FUNCTION F_RoundReal : REAL
VAR_INPUT
  rInput : REAL;
  iDecimalPlaces : INT;
END_VAR
VAR
  rOutput : REAL;
  r_Dint: DINT;
  rLeftPart : REAL;
END_VAR

rOutput := rInput * EXPT(10, iDecimalPlaces);
rLeftPart := rOutput - TRUNC(rOutput);

rOutput := TRUNC(rOutput);

IF rLeftPart >= 0.5 THEN
  	rOutput:= rOutput + 1;
ELSE
  	rOutput := rOutput;
END_IF

F_RoundReal := rOutput / EXPT(10, iDecimalPlaces);

END_FUNCTION

(* stored: Version 1.1.0.1, ProductVersion 3.1.4026.18
   POU F_RoundReal: Id {aa8a16c1-7123-4926-bb98-838e8ab366c0}, SpecialFunc None *)
